TYPE ST_System_BHKW_Stellwert :
STRUCT
	Anford_Stellventil		: BOOL;
	Anford_Pumpe		: BOOL;
	Anford_BHKW		: BOOL;
END_STRUCT
END_TYPE

(* stored: Version 1.1.0.1, ProductVersion 3.1.4024.9
   DUT ST_System_BHKW_Stellwert: Id {47ae6b6c-1d7e-4472-a600-e4f742daa1ba} *)
